// TIA Portal V16 export
// export: Created 2022-04-05T12:06:00.2185014Z, ExportSetting WithDefaults, DisplayName Totally Integrated Automation Portal, DisplayVersion V16 Update 3, DisplayName TIA Portal Version Control Interface, DisplayVersion V16 Update 2, DisplayName TIA Portal Openness, DisplayVersion V16 Update 3, DisplayName STEP 7 Professional, DisplayVersion V16 Update 3, DisplayName STEP 7 Safety, DisplayVersion V16, DisplayName WinCC Professional, DisplayVersion V16 Update 3
DATA_BLOCK "DB11001_St_DevValveIsol"   // DB11001
TITLE = Static DB [Device Driver] — Isolating Valve
{ S7_Optimized_Access := 'TRUE' }
AUTHOR : M_Gledhill
FAMILY : DeviceDriver
NAME : St_StdDevValveIsol
VERSION : 1.0
// PRACTICAL SERIES AUTOMATION LIBRARY (PAL)   —   COPYRIGHT 2020 – M. GLEDHILL (MIT LICENCE)
//                   ———— ◆ ————
//  FOR DETAILED DOCUMENTATION — SELECT THE BLOCK IN THE PROJECT TREE AND PRESS SHIFT + F1
//  FULL ONLINE DOCUMENTATION IS AVAILABLE AT: https://practicalseries.com/2001-pal/index.html
// stored: AutoNumber false, DBAccessibleFromOPCUA true, IsOnlyStoredInLoadMemory false, IsRetainMemResEnabled false, IsWriteProtectedInAS false, MemoryReserve 100
   VAR
      _DB_Header { ExternalAccessible := 'False'; ExternalVisible := 'False'; ExternalWritable := 'False'} : Array[0..79] of Bool;   // STANDARD ANALOG INSTRUMENT READ
      __________0000_0 { ExternalAccessible := 'False'; ExternalVisible := 'False'; ExternalWritable := 'False'} : Bool := false;
      __________0000_1 { ExternalAccessible := 'False'; ExternalVisible := 'False'; ExternalWritable := 'False'} : Bool := false;   // ▀▀▀▀ DB CURRENT REVISION
      revInfo { ExternalWritable := 'False'; S7_SetPoint := 'True'} : "UT01000_St_SysRevision";
      __________0010_0 { ExternalAccessible := 'False'; ExternalVisible := 'False'; ExternalWritable := 'False'} : Bool := false;
      __________0010_1 { ExternalAccessible := 'False'; ExternalVisible := 'False'; ExternalWritable := 'False'} : Bool := false;   // ▀▀▀▀ ISOLATING VALVES
      V001 { ExternalWritable := 'False'} : "UT11001_St_DevValveIsol";   // Filter 1 backwash inlet
   END_VAR
BEGIN
   // _DB_Header[0] : ▀▀▀▀▀▀▀▀▀▀▀▀▀▀▀▀▀▀▀▀▀▀▀▀▀▀▀▀▀▀▀▀▀▀▀▀▀▀▀▀▀▀▀▀
   // _DB_Header[2] : TITLE: STANDARD — DEVICE DRIVER FOR AN ISOLATING VALVE
   // _DB_Header[4] : ▄▄▄▄▄▄▄▄▄▄▄▄▄▄▄▄▄▄▄▄▄▄▄▄▄▄▄▄▄▄▄▄▄▄▄▄▄▄▄▄▄▄▄▄
   // _DB_Header[5] : TYPE: STATIC
   // _DB_Header[6] : ▀▀▀▀▀▀▀▀▀▀▀▀▀▀▀▀▀▀▀▀▀▀▀▀▀▀▀▀▀▀▀▀▀▀▀▀▀▀▀▀▀▀▀▀
   // _DB_Header[8] : This is the static data block associated with the standard device driver for an isolating valve
   // _DB_Header[9] : block:
   // _DB_Header[10] : FC11001_StdDevValveIsol
   // _DB_Header[12] : The static data holds the configuration data for the device (normally open/closed,
   // _DB_Header[13] : limit switch and interlock configuration &c.)
   // _DB_Header[15] : Each instrument is given the user data type:
   // _DB_Header[16] : UT11001_St_DevValveIsol
   // _DB_Header[17] : This holds the full set of static configuration data for the device
   // _DB_Header[19] : ━━━ ⬙⬙⬙⬙⬙⬙ ━━━
   // _DB_Header[21] : ▄▄▄▄▄▄▄▄▄▄▄▄▄▄▄▄▄▄▄▄▄▄▄▄▄▄▄▄▄▄▄▄▄▄▄▄▄▄▄▄▄▄▄▄
   // _DB_Header[22] : MODIFICATION HISTORY
   // _DB_Header[24] : This is a summary of the recent software modifications made to this block (most recent at top)
   // _DB_Header[26] : ―――――――――――――――――――――――――――――――――――――――――――
   // _DB_Header[27] : DATE REVISION MASTER BRANCH DEV
   // _DB_Header[28] : (nnn.amm) COMMIT TAG (Base ---> Merge) BRANCH Author
   // _DB_Header[29] : ———————————————————————————————————————————
   // _DB_Header[30] : 2021.08.23 001.000 D0009 D0008 D0009 None M. Gledhill
   // _DB_Header[31] : FC11001 — RELEASED FOR USE
   // _DB_Header[32] : Merge back to master branch
   // _DB_Header[34] : 2021.08.17 000.801 D0008A-000.801 D0008 N/A D0008A M. Gledhill
   // _DB_Header[35] : FC11001 Released for SMT
   // _DB_Header[37] : 2021.08.10 000.103 D0008A-000.103 D0008 N/A D0008A M. Gledhill
   // _DB_Header[38] : FC11001 Incremental build
   // _DB_Header[40] : 2021.07.21 000.102 D0008A-000.102 D0008 N/A D0008A M. Gledhill
   // _DB_Header[41] : FC11001 Incremental build
   // _DB_Header[43] : 2021.07.08 000.101 D0008A-000.101 D0008 N/A D0008A M. Gledhill
   // _DB_Header[44] : FC11001 Block created
   // _DB_Header[45] : ———————————————————————————————————————————
   // _DB_Header[46] : Where: nnn = Major revision
   // _DB_Header[47] : a = Type (1-7 Development, 8 Proving, 9 Qualification, 0 Release)
   // _DB_Header[48] : mm = Minor revision (must be 00 if a = 0)
   // _DB_Header[49] : Block properties version number should be set to nn.a (only one decimal place)
   // _DB_Header[51] : ██████████████ █ █ █ █ END █ █ █ █ ██████████████
   revInfo.REV_BLOCK := 'DB11001';
   revInfo.REV_NUMBER := '001.000';
   revInfo.REV_DATE := '2021.08.23';
   revInfo.REV_AUTHOR := 'M. Gledhill';
   V001.CONFIG_FBK_OPEN_EN := true;
   V001.CONFIG_FBK_CLOSED_EN := true;
   V001.TIME_OPENING_MAX := 20.0;
   V001.TIME_CLOSING_MAX := 30.0;
   V001.TIME_DER_OPEN := 80.0;
   V001.TIME_DER_CLOSED := 90.0;
END_DATA_BLOCK
